// TIA Portal project "GR36_BP_BeltConveyorGreen_Pro" (V17)

(* hardware
DEVICE "ET 200SP station_1"  ET 200SP-Station
   slot 0: "Rack_0"  Rack  6ES5 710-8MAx1
   slot 1: "PLC_1"  CPU 1510SP-1 PN  6ES7 510-1DJ01-0AB0  V2.1
      slot 32768: "PROFINET interface_1"  X1
   slot 2: "DI 8x24VDC HF_1"  DI 8x24VDC HF  6ES7 131-6BF00-0CA0  V2.0
      slot 1: "DI 8x24VDC HF_1"  DI 8x24VDC HF
   slot 3: "DI 8x24VDC BA_1"  DI 8x24VDC BA  6ES7 131-6BF00-0AA0  V1.0
      slot 1: "DI 8x24VDC BA_1"  DI 8x24VDC BA
   slot 4: "DQ 8x24VDC/0.5A ST_1"  DQ 8x24VDC/0.5A ST  6ES7 132-6BF00-0BA0  V1.1
      slot 1: "DQ 8x24VDC/0.5A ST_1"  DQ 8x24VDC/0.5A ST
   slot 5: "AI 2xU/I 2-,4-wire HF_1"  AI 2xU/I 2-,4-wire HF  6ES7 134-6HB00-0CA1  V2.0
      slot 1: "AI 2xU/I 2-,4-wire HF_1"  AI 2xU/I 2-,4-wire HF
   slot 6: "Server module_1"  Server module  6ES7 193-6PA00-0AA0  V1.1
      slot 1: "Server module_1"  Server module
   slot 127: "BA 2xRJ45"  BA 2xRJ45  6ES7 193-6AR00-0AA0  V0.0
      slot 32769: "Port_1"  X1 P1  6ES7 193-6AR00-0AA0
      slot 32770: "Port_2"  X1 P2  6ES7 193-6AR00-0AA0
*)

// ===== PLC "PLC_1"  CPU 1510SP-1 PN =====

VAR_GLOBAL   // PLC tag table "Default tag table"
   "Tag_14" AT %M400.0 : Bool;
   "Tag_15" AT %M400.1 : Bool;
   "Tag_16" AT %M400.2 : Bool;
   "Tag_17" AT %M400.4 : Bool;
   "Tag_18" AT %M400.5 : Bool;
   "Tag_19" AT %M400.6 : Bool;
END_VAR

VAR_GLOBAL   // PLC tag table "math"
   "mb_a1" AT %MB130 : SInt;
   "mb_a2" AT %MB131 : SInt;
   "mb_aResult" AT %MW132 : Int;
   "mb_b1" AT %MB136 : SInt;
   "md_b2" AT %MD138 : DInt;
   "mb_c1" AT %MB146 : SInt;
   "mb_c2" AT %MB147 : SInt;
   "mw_cResult" AT %MW148 : Int;
   "md_bResult" AT %MD142 : DInt;
   "mw_d1" AT %MW150 : Int;
   "mw_d2" AT %MW152 : Int;
   "md_dResult" AT %MD154 : DInt;
   "mb_e1" AT %MB158 : SInt;
   "mb_e2" AT %MB159 : SInt;
   "md_eResult" AT %MD160 : Real;
   "mw_RPM" AT %MW164 : Int;
   "mw_Gear" AT %MW166 : Int;
   "mw_DiameterShaft_mm" AT %MW168 : Int;
   "md_SpeedBelt_mm_s" AT %MD170 : Real;
END_VAR

VAR_GLOBAL   // PLC tag table "MemoryFlag_PLC"
   "m_IsBoxBetweenSensor" AT %M19.0 : Bool;
   "m_OneShoot_StartButton_Positive" AT %M20.1 : Bool;
   "m_OneShoot_StopButton_Positive" AT %M20.2 : Bool;
   "m_IsSystemON" AT %M19.1 : Bool;
   "m_AchievedMiddlePosition" AT %M19.2 : Bool;
   "m_MotorON" AT %M19.3 : Bool;
   "m_AutomaticModeON" AT %M19.4 : Bool;
   "m_OneShoot_AtMiddle_Positive" AT %M19.5 : Bool;
   "mw_CountItem" AT %MW22 : Int;
   "mw_UnsignedCount" AT %MW24 : Int;
   "mw_SlowSpeedRPM" AT %MW26 : Int;
   "mw_FastSpeedRPM" AT %MW28 : Int;
   "mb_U2Test" AT %MB40 : SInt;
   "mw_ActualSpeedRPM" AT %MW100 : Int;
   "m_OneShoot_StartButton_Negative" AT %M20.3 : Bool;
   "m_IsCoundProduct" AT %M23.2 : Bool;   // Used to detect if count is >= 4
   "m_OneShoot_ImpulsFromShaft_Positive" AT %M30.0 : Bool;
   "mw_CountImpulsFromShaft" AT %MW32 : UInt;
   "m_IsGreenLEDON" AT %M20.4 : Bool;
   "mb_CountLED" AT %MB160 : Byte;
   "m_TurnOnDelay" AT %M174.0 : Bool;
   "m_OneShoot_AtRight_Negative" AT %M200.7 : Bool;
   "m_OneShoot_AtRight_Positive" AT %M201.0 : Bool;
   "m_OneShoot_SwitchBay1_Negative" AT %M201.1 : Bool;
   "m_OneShoot_SwitchBay2_Negiative" AT %M201.2 : Bool;
   "mw_errorCode" AT %MW50 : Int;
   "TimeOut_Forward" AT %M51.0 : Bool;
   "TimeOut_Backward" AT %M51.1 : Bool;
   "IsMoreOne" AT %M51.2 : Bool;
   "m_OneShoot_AtLeft_Negative" AT %M52.0 : Bool;
END_VAR

VAR_GLOBAL   // PLC tag table "DigitalOutput_PLC"
   "dq_LedGreen" AT %Q4.0 : Bool;
   "dq_LedRed" AT %Q4.1 : Bool;
   "dq_LedWhite" AT %Q4.2 : Bool;
   "dq_LedBlue" AT %Q4.3 : Bool;
   "dqb_Lights" AT %QB4 : Byte;
END_VAR

VAR_GLOBAL   // PLC tag table "DigitalOutput_FactoryIO"
   "dq_Forward" AT %Q0.0 : Bool;
   "dq_Backward" AT %Q0.1 : Bool;
   "dq_H2" AT %Q0.3 : Bool;
   "dq_H3" AT %Q0.4 : Bool;
   "dq_Horn" AT %Q0.5 : Bool;
END_VAR

VAR_GLOBAL   // PLC tag table "DigitalInput_FactoryIO"
   "di_AtLeft_B0" AT %I0.0 : Bool;   // NO
   "di_AtMiddle_B3" AT %I0.1 : Bool;   // NC
   "di_AtRight_B5" AT %I0.2 : Bool;   // NO
   "di_FactoryIO_Running" AT %I0.7 : Bool;
   "di_ImpulsFromShaft" AT %I0.5 : Bool;
END_VAR

VAR_GLOBAL   // PLC tag table "DefultTagTable"
   "Clock_Byte" AT %MB69 : Byte;
   "Clock_10Hz" AT %M69.0 : Bool;
   "Clock_5Hz" AT %M69.1 : Bool;
   "Clock_2.5Hz" AT %M69.2 : Bool;
   "Clock_2Hz" AT %M69.3 : Bool;
   "Clock_1.25Hz" AT %M69.4 : Bool;
   "Clock_1Hz" AT %M69.5 : Bool;
   "Clock_0.625Hz" AT %M69.6 : Bool;
   "Clock_0.5Hz" AT %M69.7 : Bool;
   "System_Byte" AT %MB70 : Byte;
   "FirstScan" AT %M70.0 : Bool;
   "DiagStatusUpdate" AT %M70.1 : Bool;
   "AlwaysTRUE" AT %M70.2 : Bool;
   "AlwaysFALSE" AT %M70.3 : Bool;
   "System_Byte(1)" AT %MB1 : Byte;
   "Tag_1" AT %M10.0 : Bool;
   "Tag_2" AT %M10.1 : Bool;
   "Tag_3" AT %M20.0 : Bool;
   "Tag_4" AT %M20.7 : Bool;
   "Tag_5" AT %M21.2 : Bool;
   "Tag_6" AT %MB120 : USInt;
   "Tag_7" AT %M120.1 : Bool;
   "Tag_8" AT %M255.0 : Bool;
   "Tag_9" AT %M255.1 : Bool;
   "Tag_10" AT %M255.7 : Bool;
   "Tag_11" AT %M255.4 : Bool;
   "Tag_12" AT %M266.0 : Bool;
   "Tag_13" AT %M170.2 : Bool;
END_VAR

VAR_GLOBAL   // PLC tag table "DigitalInput_PLC"
   "di_Switch_Forward" AT %I1.0 : Bool;   // NO
   "di_Switch_Backward" AT %I1.1 : Bool;   // NO
   "di_Switch_SwitchBay1" AT %I1.2 : Bool;   // NO
   "di_Switch_SwitchBay2" AT %I1.3 : Bool;   // NO
   "di_StartButton" AT %I2.0 : Bool;   // NO
   "di_StopButton" AT %I2.1 : Bool;   // NC
   "di_Selector" AT %I2.2 : Bool;   // NO
   "di_ResetButton" AT %I2.3 : Bool;   // NC
   "dib_switch" AT %IB1 : Byte;
   "di_Switch_ResetErrors" AT %I1.7 : Bool;
   "di_Switch_ChooseSCLInBuffer" AT %I1.6 : Bool;
END_VAR

VAR_GLOBAL CONSTANT   // PLC tag table "CONST"
   "CONST_MAX_BUFFER_SIZE_LENGHT" : USInt := 9;
END_VAR

TYPE "stt_edge"
   STRUCT
      OneShoot_Positive : Bool;
      OneShoot_Negative : Bool;
      Memory : Struct
         LastState_Positive : Bool;
         LastState_Negative : Bool;
      END_STRUCT;
   END_STRUCT;
END_TYPE

DATA_BLOCK "db_mode"   // DB1
{ S7_Optimized_Access := 'TRUE' }
VERSION : 0.1
   VAR
      Manual : Bool;
      Auto : Bool;
      GlobalError : Bool;
   END_VAR
BEGIN
END_DATA_BLOCK

DATA_BLOCK "db_output"   // DB2
{ S7_Optimized_Access := 'TRUE' }
VERSION : 0.1
   VAR
      OutputManualForward : Bool;
      OutputManualBackward : Bool;
      OutputAutoForward : Bool;
      OutputAutoBackward : Bool;
   END_VAR
BEGIN
END_DATA_BLOCK

DATA_BLOCK "db_settings"   // DB3
{ S7_Optimized_Access := 'TRUE' }
VERSION : 0.1
   VAR
      goodLenght : Real := 0.45;   // The correct measurement for large pakage
      goodLenghtTolerance : Real := 0.02;
      delayResetBuffer : Time := t#4s;
      BackwardErrorDelay : Time := t#20s;
      ForwardErrorDelay : Time := t#20s;
      errorOffDelay : Time := t#3s;
      goodProductCountMAX : DInt := 4;
      conveyorSpeed : Real := 0.45;
   END_VAR
BEGIN
END_DATA_BLOCK

DATA_BLOCK "db_productInfo"   // DB4
{ S7_Optimized_Access := 'TRUE' }
VERSION : 0.1
   VAR
      "productLenght[m]" : Real;   // [m]
      maxProductLenght : Real;
      minProductLenght : Real;
      isLenghtMeasured : Bool;
      inRange : Bool;
      isProductOnConveyor : Bool;
      goodProductCount : DInt;
      productCountAfterAtLeft : DInt;
      isProductInLine : Word;
      isProductCountExceeded : Bool;
      timeStamp : DTL;
      label : String;
      maxValueInBufforArray : Real;
   END_VAR
BEGIN
END_DATA_BLOCK

DATA_BLOCK "db_buffor"   // DB7
{ S7_Optimized_Access := 'TRUE' }
VERSION : 0.1
   VAR RETAIN
      IndexOfArray_Lenght : USInt := 3;
      Lenght : Array[0.."CONST_MAX_BUFFER_SIZE_LENGHT"] of Real;
   END_VAR
BEGIN
   Lenght[0] := 0.2772;
   Lenght[1] := 0.2646;
   Lenght[2] := 0.26505;
   Lenght[3] := 0.42255;
   Lenght[4] := 0.42255;
   Lenght[5] := 0.42255;
   Lenght[6] := 0.42255;
   Lenght[7] := 0.42255;
   Lenght[8] := 0.42255;
   Lenght[9] := 0.0;
END_DATA_BLOCK

DATA_BLOCK "db_edge"   // DB11
{ S7_Optimized_Access := 'TRUE' }
VERSION : 0.1
   VAR
      SwitchForward : "stt_edge";
      AtRight : "stt_edge";
      AtLeft : "stt_edge";
      AtMiddle : "stt_edge";
      SwitchBay1 : "stt_edge";
      SwitchBay2 : "stt_edge";
   END_VAR
BEGIN
END_DATA_BLOCK

// folder: System blocks/Program resources

DATA_BLOCK "tonr_accumulateAtMiddleTravelsalTime"   // DB5
{ S7_Optimized_Access := 'TRUE' }
AUTHOR : Simatic
FAMILY : IEC
NAME : IEC_TMR
VERSION : 1.0
// stored: InstanceOfName IEC_TIMER
"IEC_TIMER"
BEGIN
END_DATA_BLOCK

DATA_BLOCK "ton_resetButtonHowLong"   // DB6
{ S7_Optimized_Access := 'TRUE' }
AUTHOR : Simatic
FAMILY : IEC
NAME : IEC_TMR
VERSION : 1.0
// stored: InstanceOfName IEC_TIMER
"IEC_TIMER"
BEGIN
END_DATA_BLOCK

DATA_BLOCK "ctu_errorSignalization"   // DB9
{ S7_Optimized_Access := 'TRUE' }
AUTHOR : Simatic
FAMILY : IEC
NAME : CNTR
VERSION : 1.0
// stored: InstanceOfName IEC_COUNTER
"IEC_COUNTER"
BEGIN
END_DATA_BLOCK

DATA_BLOCK "ton_errorLedOffDelay"   // DB10
{ S7_Optimized_Access := 'TRUE' }
AUTHOR : Simatic
FAMILY : IEC
NAME : IEC_TMR
VERSION : 1.0
// stored: InstanceOfName IEC_TIMER
"IEC_TIMER"
BEGIN
END_DATA_BLOCK

// folder: (top level)

FUNCTION "fc_mode" : Void   // FC1, LAD
{ S7_Optimized_Access := 'TRUE' }
VERSION : 0.1
BEGIN

REGION Network 1: Turn on manual mode
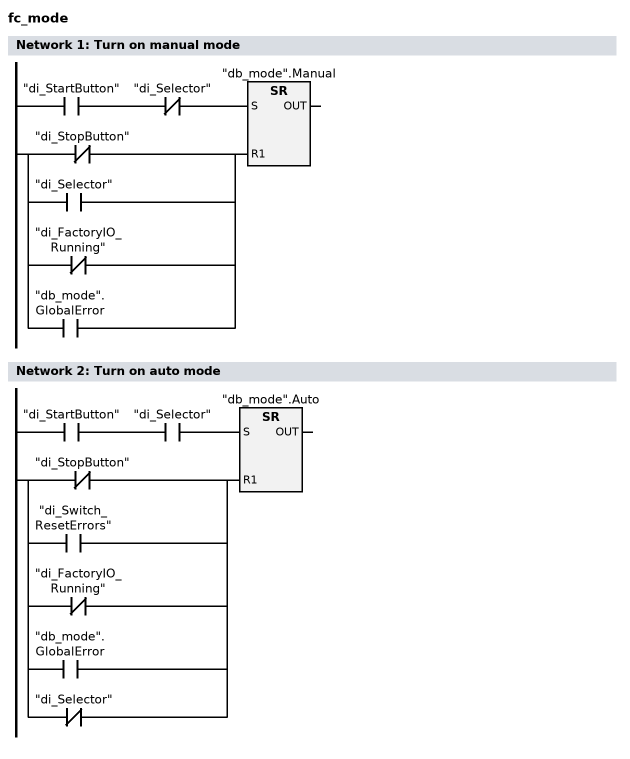
   RUNG wire#powerrail
      Contact( "di_StartButton" )
      I_Contact( "di_Selector" )
      S_SR(operand := "db_mode".Manual, r1 := wire#w1)
   END_RUNG
   RUNG wire#powerrail
      I_Contact( "di_StopButton" )
   END_RUNG wire#w1
   RUNG wire#powerrail
      Contact( "di_Selector" )
   END_RUNG wire#w1
   RUNG wire#powerrail
      I_Contact( "di_FactoryIO_Running" )
   END_RUNG wire#w1
   RUNG wire#powerrail
      Contact( "db_mode".GlobalError )
   END_RUNG wire#w1
   // the same network as SCL:
   IF "di_StartButton" AND NOT "di_Selector" THEN
       "db_mode".Manual := TRUE;   // SR flip-flop
   END_IF;
   IF NOT "di_StopButton" OR "di_Selector" OR NOT "di_FactoryIO_Running" OR "db_mode".GlobalError THEN
       "db_mode".Manual := FALSE;
   END_IF;
END_REGION

REGION Network 2: Turn on auto mode
   RUNG wire#powerrail
      Contact( "di_StartButton" )
      Contact( "di_Selector" )
      S_SR(operand := "db_mode".Auto, r1 := wire#w1)
   END_RUNG
   RUNG wire#powerrail
      I_Contact( "di_StopButton" )
   END_RUNG wire#w1
   RUNG wire#powerrail
      Contact( "di_Switch_ResetErrors" )
   END_RUNG wire#w1
   RUNG wire#powerrail
      I_Contact( "di_FactoryIO_Running" )
   END_RUNG wire#w1
   RUNG wire#powerrail
      Contact( "db_mode".GlobalError )
   END_RUNG wire#w1
   RUNG wire#powerrail
      I_Contact( "di_Selector" )
   END_RUNG wire#w1
   // the same network as SCL:
   IF "di_StartButton" AND "di_Selector" THEN
       "db_mode".Auto := TRUE;   // SR flip-flop
   END_IF;
   IF NOT "di_StopButton" OR "di_Switch_ResetErrors" OR NOT "di_FactoryIO_Running" OR "db_mode".GlobalError OR NOT "di_Selector" THEN
       "db_mode".Auto := FALSE;
   END_IF;
END_REGION
END_FUNCTION

FUNCTION "fc_manual" : Void   // FC2, LAD
{ S7_Optimized_Access := 'TRUE' }
VERSION : 0.1
BEGIN

REGION Network 1: Moving forward
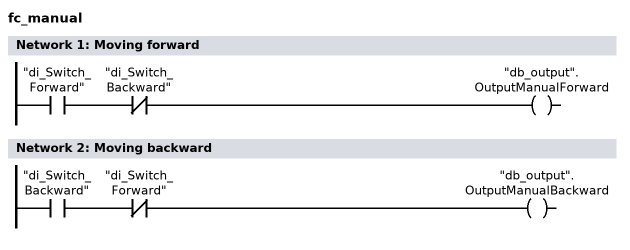
   RUNG wire#powerrail
      Contact( "di_Switch_Forward" )
      I_Contact( "di_Switch_Backward" )
      Coil( "db_output".OutputManualForward )
   END_RUNG
   // the same network as SCL:
   "db_output".OutputManualForward := "di_Switch_Forward" AND NOT "di_Switch_Backward";
END_REGION

REGION Network 2: Moving backward
   RUNG wire#powerrail
      Contact( "di_Switch_Backward" )
      I_Contact( "di_Switch_Forward" )
      Coil( "db_output".OutputManualBackward )
   END_RUNG
   // the same network as SCL:
   "db_output".OutputManualBackward := "di_Switch_Backward" AND NOT "di_Switch_Forward";
END_REGION
END_FUNCTION

FUNCTION "fc_auto" : Void   // FC3, LAD
{ S7_Optimized_Access := 'TRUE' }
VERSION : 0.1
   VAR_TEMP
      temp_LSB : Word;
   END_VAR
BEGIN

REGION Network 1: Move forward
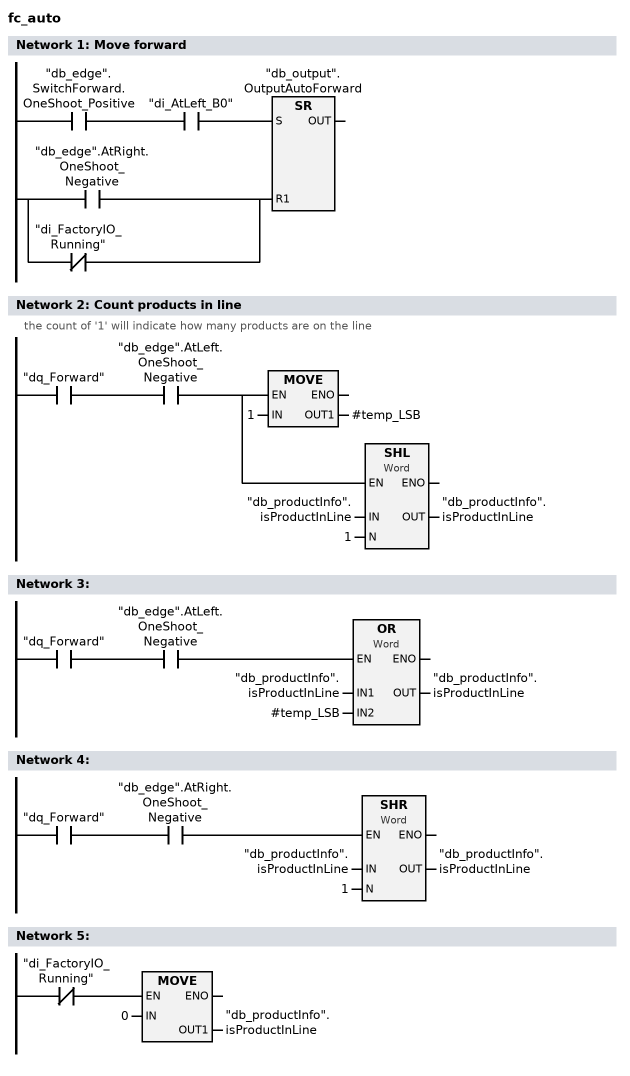
   RUNG wire#powerrail
      Contact( "db_edge".SwitchForward.OneShoot_Positive )
      Contact( "di_AtLeft_B0" )
      S_SR(operand := "db_output".OutputAutoForward, r1 := wire#w1)
   END_RUNG
   RUNG wire#powerrail
      Contact( "db_edge".AtRight.OneShoot_Negative )
   END_RUNG wire#w1
   RUNG wire#powerrail
      I_Contact( "di_FactoryIO_Running" )
   END_RUNG wire#w1
   // the same network as SCL:
   IF "db_edge".SwitchForward.OneShoot_Positive AND "di_AtLeft_B0" THEN
       "db_output".OutputAutoForward := TRUE;   // SR flip-flop
   END_IF;
   IF "db_edge".AtRight.OneShoot_Negative OR NOT "di_FactoryIO_Running" THEN
       "db_output".OutputAutoForward := FALSE;
   END_IF;
END_REGION

REGION Network 2: Count products in line
   // the count of '1' will indicate how many products are on the line
   RUNG wire#powerrail
      Contact( "dq_Forward" )
      Contact( "db_edge".AtLeft.OneShoot_Negative )
      wire#w1
      Move(in := 1, out1 => #temp_LSB)
   END_RUNG
   RUNG wire#w1
      { S7_Templates := "SrcType := Word" } Shl(in := "db_productInfo".isProductInLine, n := 1, out => "db_productInfo".isProductInLine)
   END_RUNG
   // the same network as SCL:
   IF "dq_Forward" AND "db_edge".AtLeft.OneShoot_Negative THEN
       #temp_LSB := 1;
       "db_productInfo".isProductInLine := SHL(IN := "db_productInfo".isProductInLine, N := 1);
   END_IF;
END_REGION

REGION Network 3
   IF "dq_Forward" AND "db_edge".AtLeft.OneShoot_Negative THEN
       "db_productInfo".isProductInLine := "db_productInfo".isProductInLine OR #temp_LSB;
   END_IF;
END_REGION

REGION Network 4
   RUNG wire#powerrail
      Contact( "dq_Forward" )
      Contact( "db_edge".AtRight.OneShoot_Negative )
      { S7_Templates := "SrcType := Word" } Shr(in := "db_productInfo".isProductInLine, n := 1, out => "db_productInfo".isProductInLine)
   END_RUNG
   // the same network as SCL:
   IF "dq_Forward" AND "db_edge".AtRight.OneShoot_Negative THEN
       "db_productInfo".isProductInLine := SHR(IN := "db_productInfo".isProductInLine, N := 1);
   END_IF;
END_REGION

REGION Network 5
   RUNG wire#powerrail
      I_Contact( "di_FactoryIO_Running" )
      Move(in := 0, out1 => "db_productInfo".isProductInLine)
   END_RUNG
   // the same network as SCL:
   IF NOT "di_FactoryIO_Running" THEN "db_productInfo".isProductInLine := 0; END_IF;
END_REGION
END_FUNCTION

FUNCTION "fc_output" : Void   // FC4, LAD
{ S7_Optimized_Access := 'TRUE' }
VERSION : 0.1
BEGIN

REGION Network 1: Handle moving forward
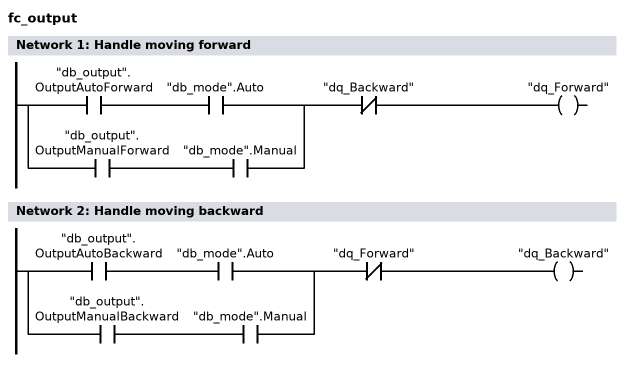
   RUNG wire#powerrail
      Contact( "db_output".OutputAutoForward )
      Contact( "db_mode".Auto )
      wire#w1
      I_Contact( "dq_Backward" )
      Coil( "dq_Forward" )
   END_RUNG
   RUNG wire#powerrail
      Contact( "db_output".OutputManualForward )
      Contact( "db_mode".Manual )
   END_RUNG wire#w1
   // the same network as SCL:
   "dq_Forward" := (("db_output".OutputAutoForward AND "db_mode".Auto) OR ("db_output".OutputManualForward AND "db_mode".Manual)) AND NOT "dq_Backward";
END_REGION

REGION Network 2: Handle moving backward
   RUNG wire#powerrail
      Contact( "db_output".OutputAutoBackward )
      Contact( "db_mode".Auto )
      wire#w1
      I_Contact( "dq_Forward" )
      Coil( "dq_Backward" )
   END_RUNG
   RUNG wire#powerrail
      Contact( "db_output".OutputManualBackward )
      Contact( "db_mode".Manual )
   END_RUNG wire#w1
   // the same network as SCL:
   "dq_Backward" := (("db_output".OutputAutoBackward AND "db_mode".Auto) OR ("db_output".OutputManualBackward AND "db_mode".Manual)) AND NOT "dq_Forward";
END_REGION
END_FUNCTION

FUNCTION "fc_lightSoundSignalization" : Void   // FC5, LAD
{ S7_Optimized_Access := 'TRUE' }
VERSION : 0.1
   VAR_TEMP   // added for the SCL form of the ladder/FBD networks
      _w1 : Bool;
   END_VAR
BEGIN

REGION Network 1: Light mode signalization
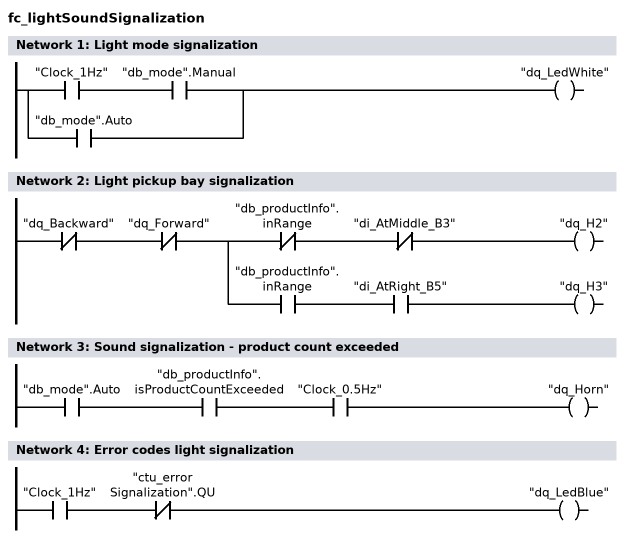
   RUNG wire#powerrail
      Contact( "Clock_1Hz" )
      Contact( "db_mode".Manual )
      wire#w1
      Coil( "dq_LedWhite" )
   END_RUNG
   RUNG wire#powerrail
      Contact( "db_mode".Auto )
   END_RUNG wire#w1
   // the same network as SCL:
   "dq_LedWhite" := ("Clock_1Hz" AND "db_mode".Manual) OR "db_mode".Auto;
END_REGION

REGION Network 2: Light pickup bay signalization
   RUNG wire#powerrail
      I_Contact( "dq_Backward" )
      I_Contact( "dq_Forward" )
      wire#w1
      I_Contact( "db_productInfo".inRange )
      I_Contact( "di_AtMiddle_B3" )
      Coil( "dq_H2" )
   END_RUNG
   RUNG wire#w1
      Contact( "db_productInfo".inRange )
      Contact( "di_AtRight_B5" )
      Coil( "dq_H3" )
   END_RUNG
   // the same network as SCL:
   #_w1 := NOT "dq_Backward" AND NOT "dq_Forward";
   "dq_H2" := #_w1 AND NOT "db_productInfo".inRange AND NOT "di_AtMiddle_B3";
   "dq_H3" := #_w1 AND "db_productInfo".inRange AND "di_AtRight_B5";
END_REGION

REGION Network 3: Sound signalization - product count exceeded
   RUNG wire#powerrail
      Contact( "db_mode".Auto )
      Contact( "db_productInfo".isProductCountExceeded )
      Contact( "Clock_0.5Hz" )
      Coil( "dq_Horn" )
   END_RUNG
   // the same network as SCL:
   "dq_Horn" := "db_mode".Auto AND "db_productInfo".isProductCountExceeded AND "Clock_0.5Hz";
END_REGION

REGION Network 4: Error codes light signalization
   RUNG wire#powerrail
      Contact( "Clock_1Hz" )
      I_Contact( "ctu_errorSignalization".QU )
      Coil( "dq_LedBlue" )
   END_RUNG
   // the same network as SCL:
   "dq_LedBlue" := "Clock_1Hz" AND NOT "ctu_errorSignalization".QU;
END_REGION
END_FUNCTION

FUNCTION "fc_sizeOfProduct" : Void   // FC6, LAD
{ S7_Optimized_Access := 'TRUE' }
VERSION : 0.1
   VAR_TEMP
      temp_travelsalTime : DInt;
   END_VAR
BEGIN

REGION Network 1: Get the time of travesal through right sensor
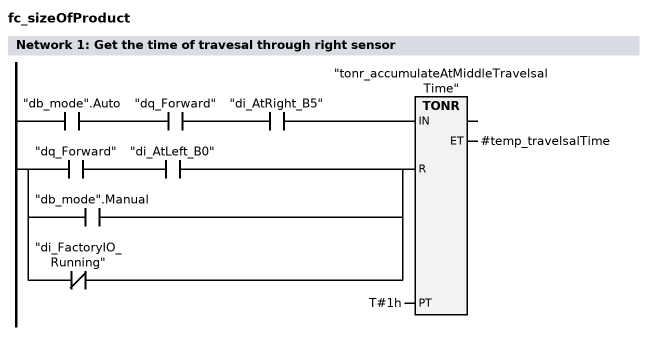
   "tonr_accumulateAtMiddleTravelsalTime".TONR(IN := "db_mode".Auto AND "dq_Forward" AND "di_AtRight_B5",
                           R := ("dq_Forward" AND "di_AtLeft_B0") OR "db_mode".Manual OR NOT "di_FactoryIO_Running",
                           PT := T#1h,
                           ET => #temp_travelsalTime);
END_REGION

REGION Network 2 (SCL): Calculate package lenght (result in [m])
   // Caluclate current package lenght
   "db_productInfo"."productLenght[m]" := "db_settings".conveyorSpeed * DINT_TO_REAL(#temp_travelsalTime) / 1000.0;

   // Calculate boundaries for package lenght
   "db_productInfo".maxProductLenght := "db_settings".goodLenght + "db_settings".goodLenghtTolerance;
   "db_productInfo".minProductLenght := "db_settings".goodLenght - "db_settings".goodLenghtTolerance;
END_REGION
END_FUNCTION

FUNCTION "fc_edge" : Void   // FC7, LAD
TITLE = Detect pos and neg edge
{ S7_Optimized_Access := 'TRUE' }
VERSION : 0.1
   VAR_TEMP   // added for the SCL form of the ladder/FBD networks
      _w1 : Bool;
      _w2 : Bool;
   END_VAR
BEGIN

REGION Network 1: AtRight
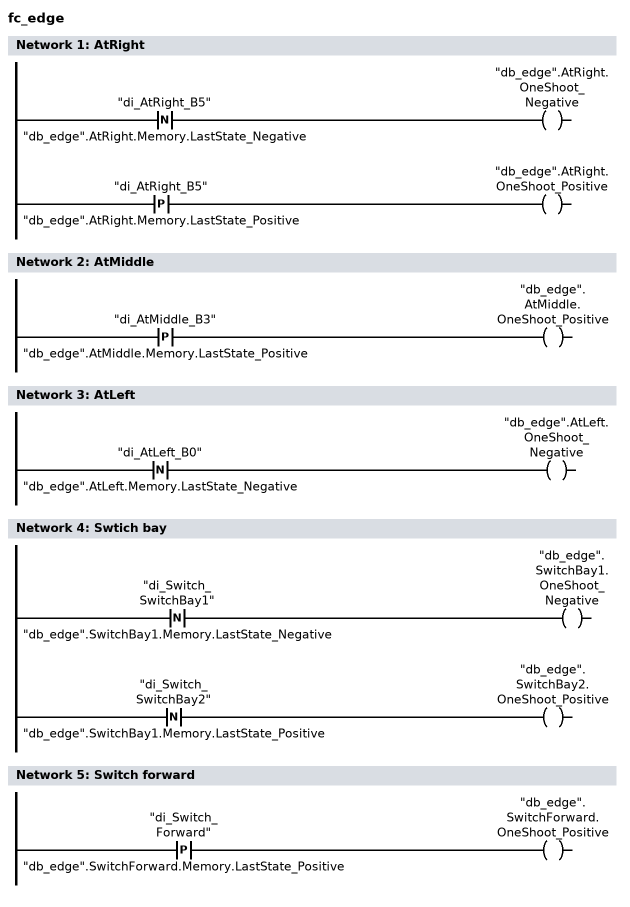
   RUNG wire#powerrail
      N_Contact(operand := "di_AtRight_B5", bit := "db_edge".AtRight.Memory.LastState_Negative)
      Coil( "db_edge".AtRight.OneShoot_Negative )
   END_RUNG
   RUNG wire#powerrail
      P_Contact(operand := "di_AtRight_B5", bit := "db_edge".AtRight.Memory.LastState_Positive)
      Coil( "db_edge".AtRight.OneShoot_Positive )
   END_RUNG
   // the same network as SCL:
   #_w1 := NOT "di_AtRight_B5" AND "db_edge".AtRight.Memory.LastState_Negative;   // falling edge of "di_AtRight_B5"
   "db_edge".AtRight.Memory.LastState_Negative := "di_AtRight_B5";
   "db_edge".AtRight.OneShoot_Negative := #_w1;
   #_w2 := "di_AtRight_B5" AND NOT "db_edge".AtRight.Memory.LastState_Positive;   // rising edge of "di_AtRight_B5"
   "db_edge".AtRight.Memory.LastState_Positive := "di_AtRight_B5";
   "db_edge".AtRight.OneShoot_Positive := #_w2;
END_REGION

REGION Network 2: AtMiddle
   RUNG wire#powerrail
      P_Contact(operand := "di_AtMiddle_B3", bit := "db_edge".AtMiddle.Memory.LastState_Positive)
      Coil( "db_edge".AtMiddle.OneShoot_Positive )
   END_RUNG
   // the same network as SCL:
   #_w1 := "di_AtMiddle_B3" AND NOT "db_edge".AtMiddle.Memory.LastState_Positive;   // rising edge of "di_AtMiddle_B3"
   "db_edge".AtMiddle.Memory.LastState_Positive := "di_AtMiddle_B3";
   "db_edge".AtMiddle.OneShoot_Positive := #_w1;
END_REGION

REGION Network 3: AtLeft
   RUNG wire#powerrail
      N_Contact(operand := "di_AtLeft_B0", bit := "db_edge".AtLeft.Memory.LastState_Negative)
      Coil( "db_edge".AtLeft.OneShoot_Negative )
   END_RUNG
   // the same network as SCL:
   #_w1 := NOT "di_AtLeft_B0" AND "db_edge".AtLeft.Memory.LastState_Negative;   // falling edge of "di_AtLeft_B0"
   "db_edge".AtLeft.Memory.LastState_Negative := "di_AtLeft_B0";
   "db_edge".AtLeft.OneShoot_Negative := #_w1;
END_REGION

REGION Network 4: Swtich bay
   RUNG wire#powerrail
      N_Contact(operand := "di_Switch_SwitchBay1", bit := "db_edge".SwitchBay1.Memory.LastState_Negative)
      Coil( "db_edge".SwitchBay1.OneShoot_Negative )
   END_RUNG
   RUNG wire#powerrail
      N_Contact(operand := "di_Switch_SwitchBay2", bit := "db_edge".SwitchBay1.Memory.LastState_Positive)
      Coil( "db_edge".SwitchBay2.OneShoot_Positive )
   END_RUNG
   // the same network as SCL:
   #_w1 := NOT "di_Switch_SwitchBay1" AND "db_edge".SwitchBay1.Memory.LastState_Negative;   // falling edge of "di_Switch_SwitchBay1"
   "db_edge".SwitchBay1.Memory.LastState_Negative := "di_Switch_SwitchBay1";
   "db_edge".SwitchBay1.OneShoot_Negative := #_w1;
   #_w2 := NOT "di_Switch_SwitchBay2" AND "db_edge".SwitchBay1.Memory.LastState_Positive;   // falling edge of "di_Switch_SwitchBay2"
   "db_edge".SwitchBay1.Memory.LastState_Positive := "di_Switch_SwitchBay2";
   "db_edge".SwitchBay2.OneShoot_Positive := #_w2;
END_REGION

REGION Network 5: Switch forward
   RUNG wire#powerrail
      P_Contact(operand := "di_Switch_Forward", bit := "db_edge".SwitchForward.Memory.LastState_Positive)
      Coil( "db_edge".SwitchForward.OneShoot_Positive )
   END_RUNG
   // the same network as SCL:
   #_w1 := "di_Switch_Forward" AND NOT "db_edge".SwitchForward.Memory.LastState_Positive;   // rising edge of "di_Switch_Forward"
   "db_edge".SwitchForward.Memory.LastState_Positive := "di_Switch_Forward";
   "db_edge".SwitchForward.OneShoot_Positive := #_w1;
END_REGION
END_FUNCTION

FUNCTION "fc_countProducts" : Void   // FC8, LAD
{ S7_Optimized_Access := 'TRUE' }
VERSION : 0.1
   VAR_TEMP   // added for the SCL form of the ladder/FBD networks
      _w1 : Bool;
   END_VAR
BEGIN

REGION Network 1: Count transported products
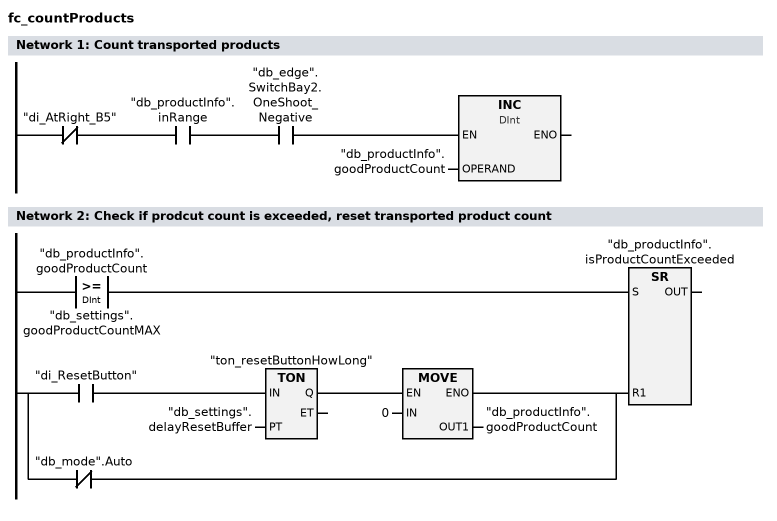
   RUNG wire#powerrail
      I_Contact( "di_AtRight_B5" )
      Contact( "db_productInfo".inRange )
      Contact( "db_edge".SwitchBay2.OneShoot_Negative )
      { S7_Templates := "DestType := DInt" } Inc( "db_productInfo".goodProductCount )
   END_RUNG
   // the same network as SCL:
   IF NOT "di_AtRight_B5" AND "db_productInfo".inRange AND "db_edge".SwitchBay2.OneShoot_Negative THEN
       "db_productInfo".goodProductCount := "db_productInfo".goodProductCount + 1;
   END_IF;
END_REGION

REGION Network 2: Check if prodcut count is exceeded, reset transported product count
   "ton_resetButtonHowLong".TON(IN := "di_ResetButton", PT := "db_settings".delayResetBuffer);
   #_w1 := "db_productInfo".goodProductCount >= "db_settings".goodProductCountMAX;
   IF "ton_resetButtonHowLong".Q THEN "db_productInfo".goodProductCount := 0; END_IF;
   IF #_w1 THEN
       "db_productInfo".isProductCountExceeded := TRUE;   // SR flip-flop
   END_IF;
   IF "ton_resetButtonHowLong".Q OR NOT "db_mode".Auto THEN
       "db_productInfo".isProductCountExceeded := FALSE;
   END_IF;
END_REGION
END_FUNCTION

FUNCTION "fc_error" : Void   // FC9, LAD
{ S7_Optimized_Access := 'TRUE' }
VERSION : 0.1
BEGIN

REGION Network 1: Global error
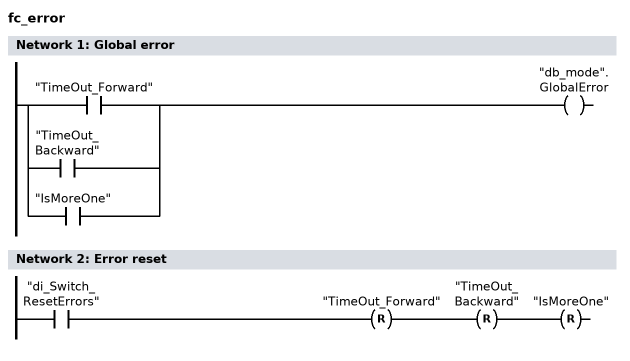
   RUNG wire#powerrail
      Contact( "TimeOut_Forward" )
      wire#w1
      Coil( "db_mode".GlobalError )
   END_RUNG
   RUNG wire#powerrail
      Contact( "TimeOut_Backward" )
   END_RUNG wire#w1
   RUNG wire#powerrail
      Contact( "IsMoreOne" )
   END_RUNG wire#w1
   // the same network as SCL:
   "db_mode".GlobalError := "TimeOut_Forward" OR "TimeOut_Backward" OR "IsMoreOne";
END_REGION

REGION Network 2: Error reset
   RUNG wire#powerrail
      Contact( "di_Switch_ResetErrors" )
      R_Coil( "TimeOut_Forward" )
      R_Coil( "TimeOut_Backward" )
      R_Coil( "IsMoreOne" )
   END_RUNG
   // the same network as SCL:
   IF "di_Switch_ResetErrors" THEN
       "TimeOut_Forward" := FALSE;
       "TimeOut_Backward" := FALSE;
       "IsMoreOne" := FALSE;
   END_IF;
END_REGION
END_FUNCTION

FUNCTION "fc_codeGenerator" : Void   // FC10, LAD
{ S7_Optimized_Access := 'TRUE' }
VERSION : 0.1
BEGIN

REGION Network 1: Generate Blue LED signal to signal error codes
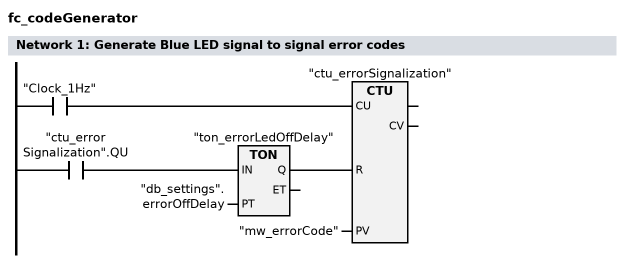
   "ton_errorLedOffDelay".TON(IN := "ctu_errorSignalization".QU, PT := "db_settings".errorOffDelay);
   "ctu_errorSignalization".CTU(CU := "Clock_1Hz", R := "ton_errorLedOffDelay".Q, PV := "mw_errorCode");
END_REGION
END_FUNCTION

FUNCTION "fc_buffor" : Void   // FC11, LAD
TITLE = Stores product lenghts in an buffer
{ S7_Optimized_Access := 'TRUE' }
VERSION : 0.1
   VAR_TEMP
      temp_arrayBufforIndex : USInt;
   END_VAR
BEGIN

REGION Network 1 (SCL): Store lenght of products in a buffer
   // Check if product has left the conveyor   
   IF "dq_Forward" AND "db_edge".AtRight.OneShoot_Negative THEN

       // Store i-th lenght in an array
       "db_buffor".Lenght["db_buffor".IndexOfArray_Lenght] := "db_productInfo"."productLenght[m]";

       // Increse the index vaiable, if exceedes max lenght set it to 0
       "db_buffor".IndexOfArray_Lenght := "db_buffor".IndexOfArray_Lenght + 1;

       IF "db_buffor".IndexOfArray_Lenght >= "CONST_MAX_BUFFER_SIZE_LENGHT" THEN
           "db_buffor".IndexOfArray_Lenght := 0;
       END_IF;
   END_IF;
END_REGION

REGION Network 2: Ladder approach to find max value
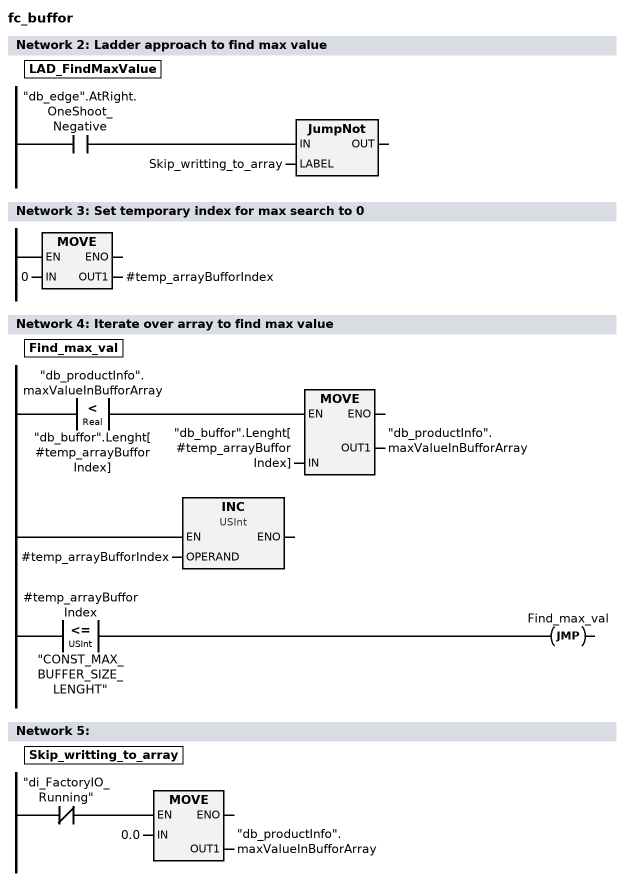
   // no SCL statement known for JumpNot: written as a call
   LAD_FindMaxValue:
   JumpNot(in := "db_edge".AtRight.OneShoot_Negative, label := Skip_writting_to_array);
END_REGION

REGION Network 3: Set temporary index for max search to 0
   RUNG wire#powerrail
      Move(in := 0, out1 => #temp_arrayBufforIndex)
   END_RUNG
   // the same network as SCL:
   #temp_arrayBufforIndex := 0;
END_REGION

REGION Network 4: Iterate over array to find max value
   Label( Find_max_val )
   RUNG wire#powerrail
      { S7_Templates := "SrcType := Real" } LT_Contact(in1 := "db_productInfo".maxValueInBufforArray, in2 := "db_buffor".Lenght[#temp_arrayBufforIndex])
      Move(in := "db_buffor".Lenght[#temp_arrayBufforIndex], out1 => "db_productInfo".maxValueInBufforArray)
   END_RUNG
   RUNG wire#powerrail
      { S7_Templates := "DestType := USInt" } Inc( #temp_arrayBufforIndex )
   END_RUNG
   RUNG wire#powerrail
      { S7_Templates := "SrcType := USInt" } LE_Contact(in1 := #temp_arrayBufforIndex, in2 := "CONST_MAX_BUFFER_SIZE_LENGHT")
      JumpCoil( Find_max_val )
   END_RUNG
   // the same network as SCL:
   Find_max_val:
   IF "db_productInfo".maxValueInBufforArray < "db_buffor".Lenght[#temp_arrayBufforIndex] THEN
       "db_productInfo".maxValueInBufforArray := "db_buffor".Lenght[#temp_arrayBufforIndex];
   END_IF;
   #temp_arrayBufforIndex := #temp_arrayBufforIndex + 1;
   IF #temp_arrayBufforIndex <= "CONST_MAX_BUFFER_SIZE_LENGHT" THEN GOTO Find_max_val; END_IF;
END_REGION

REGION Network 5
   Label( Skip_writting_to_array )
   RUNG wire#powerrail
      I_Contact( "di_FactoryIO_Running" )
      Move(in := 0.0, out1 => "db_productInfo".maxValueInBufforArray)
   END_RUNG
   // the same network as SCL:
   Skip_writting_to_array:
   IF NOT "di_FactoryIO_Running" THEN "db_productInfo".maxValueInBufforArray := 0.0; END_IF;
END_REGION
END_FUNCTION

FUNCTION "fc_buffor_scl" : Void   // FC12, LAD
{ S7_Optimized_Access := 'TRUE' }
VERSION : 0.1
   VAR_TEMP
      temp_arrayBufforIndex : USInt;
   END_VAR
BEGIN

REGION Network 1 (SCL): Store lenght of products in a buffer
   // Check if product has left the conveyor   
   IF "dq_Forward" AND "db_edge".AtRight.OneShoot_Negative THEN

       // Store i-th lenght in an array
       "db_buffor".Lenght["db_buffor".IndexOfArray_Lenght] := "db_productInfo"."productLenght[m]";

       // Increse the index vaiable, if exceedes max lenght set it to 0
       "db_buffor".IndexOfArray_Lenght := "db_buffor".IndexOfArray_Lenght + 1;

       IF "db_buffor".IndexOfArray_Lenght >= "CONST_MAX_BUFFER_SIZE_LENGHT" THEN
           "db_buffor".IndexOfArray_Lenght := 0;
       END_IF;
   END_IF;
END_REGION

REGION Network 2 (SCL): Find max value in the array
   IF "dq_Forward" AND "db_edge".AtRight.OneShoot_Negative THEN

       FOR #temp_arrayBufforIndex := 0 TO "CONST_MAX_BUFFER_SIZE_LENGHT" DO

           IF "db_buffor".Lenght[#temp_arrayBufforIndex] > "db_productInfo".maxValueInBufforArray THEN
               "db_productInfo".maxValueInBufforArray := "db_buffor".Lenght[#temp_arrayBufforIndex];
           END_IF;
       END_FOR;
   END_IF;
END_REGION
END_FUNCTION

ORGANIZATION_BLOCK "Main"   // OB1, LAD, ProgramCycle
TITLE = "Main Program Sweep (Cycle)"
{ S7_Optimized_Access := 'TRUE' }
VERSION : 0.1
   VAR_INPUT
      Initial_Call : Bool;   // Initial call of this OB
      Remanence : Bool;   // =True, if remanent data are available
   END_VAR
BEGIN

REGION Network 1: Call funcitons
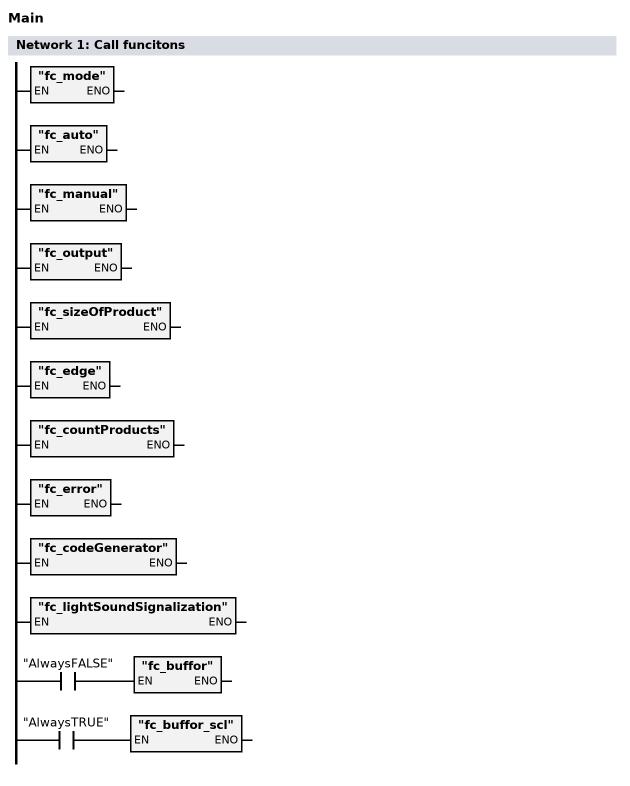
   RUNG wire#powerrail
      "fc_mode"()
   END_RUNG
   RUNG wire#powerrail
      "fc_auto"()
   END_RUNG
   RUNG wire#powerrail
      "fc_manual"()
   END_RUNG
   RUNG wire#powerrail
      "fc_output"()
   END_RUNG
   RUNG wire#powerrail
      "fc_sizeOfProduct"()
   END_RUNG
   RUNG wire#powerrail
      "fc_edge"()
   END_RUNG
   RUNG wire#powerrail
      "fc_countProducts"()
   END_RUNG
   RUNG wire#powerrail
      "fc_error"()
   END_RUNG
   RUNG wire#powerrail
      "fc_codeGenerator"()
   END_RUNG
   RUNG wire#powerrail
      "fc_lightSoundSignalization"()
   END_RUNG
   RUNG wire#powerrail
      Contact( "AlwaysFALSE" )
      "fc_buffor"()
   END_RUNG
   RUNG wire#powerrail
      Contact( "AlwaysTRUE" )
      "fc_buffor_scl"()
   END_RUNG
   // the same network as SCL:
   "fc_mode"();
   "fc_auto"();
   "fc_manual"();
   "fc_output"();
   "fc_sizeOfProduct"();
   "fc_edge"();
   "fc_countProducts"();
   "fc_error"();
   "fc_codeGenerator"();
   "fc_lightSoundSignalization"();
   IF "AlwaysFALSE" THEN "fc_buffor"(); END_IF;
   IF "AlwaysTRUE" THEN "fc_buffor_scl"(); END_IF;
END_REGION
END_ORGANIZATION_BLOCK